// SIMATIC S7-200 project (STEP 7-Micro/WIN), CPU 224 REL 02.00

ORGANIZATION_BLOCK 主程序:OB1
TITLE=---|基于 S7-200 PLC 的步进电机控制系统|---
// 设备启动时，程序利用程序启动标志初始化脉冲输出参数，包括脉冲周期500μs和最大步数429496700。用户可以通过旋转方向开关选择电机的旋转方向，并由电机方向控制输出信号控制（1=逆时针，0=顺时针），但只有在电机停止时，才能改变旋转方向，以确保运行中的稳定性。系统配备了启动按钮和停止按钮来控制电机的运行。按下启动按钮时，若无联锁、电机停止且步数大于1，则通过脉冲输出控制寄存器启动脉冲输出，电机开始运动，同时置位电机运行标志。需要注意的是，脉冲输出的步数必须大于1才能启动电机，以保证有效操作。
// 按下停止按钮后，系统调用停止电机子程序停止脉冲输出并复位标志，同时激活联锁，需松开启动按钮才能解除联锁，确保操作安全。用户还可以通过设置参考点按钮初始化电机位置。按下该按钮时，若电机正在运行，系统会先停止电机，然后通过操作模式选择子程序设置参考点并切换模式。在电机运行时，操作模式保持不变，以维持当前任务的顺利进行。
// 参考点设置完成后，定位控制激活指示点亮，系统进入定位控制模式。此时，用户输入定位角度，定位控制子程序根据角度计算步数（角度/9 * 25 + 余数调整），并由步数调整子程序微调步数，确保定位精度。只有在参考点已设置后，才能执行定位控制，以保证定位的准确性。当脉冲输出完成时，脉冲中止中断自动触发，复位电机运行标志，确保电机及时停止并避免超程。
BEGIN
Network 1 // 网络标题
// 用脉冲输出进行定位控制
LD     SM0.1
R      M0.0, 128             //M0.0 至MD12复位
ATCH   INT_0:INT0, 19
//把中断0分配给中断事件19 (脉冲串终止)
ENI
//脉冲输出功能初始化
MOVW   500, SMW68            //脉冲周期T=500US
MOVW   0, SMW70              // 脉冲宽度为0(脉冲调制)
MOVD   429496700, SMD72      //为参考点设定最大脉冲数
//设置逆时针旋转
LDN    M0.1                  //若电机停止
A      I1.5                  //且旋转主向开关=1 
S      Q0.2, 1               //则逆时针旋转
//设置顺时针旋转
LDN    M0.1                  //若电机停止
AN     I1.5                  //且旋转方向开关=0
R      Q0.2, 1               //则逆时针旋转(Q0.2=0)
//联锁
LD     I1.1
//若按"STOP"(停止)按钮
S      M0.2, 1               //则激活联锁
//解除联锁                   //
LDN    I1.1                  //且"STOP"(停止)按钮松开
AN     I1.0                  //若"START"(启动)按钮松开
R      M0.2, 1               //解除联锁
//确定操作模式(参考点定位控制)
LD     I1.4                  //若按"设置参考点"按钮
EU                           //上升沿
CALL   SBR_1:SBR1
//启动电机
LD     I1.0
// 若按"START"(启动)按钮
EU                           //上升沿
AN     M0.1                  //且电机停止
AN     M0.2                  // 且无联锁
AD>=   SMD72, 1              //且;步数大于1
MOVB   16#85, SMB67          //置脉冲输出功能(PTO)的控制位
PLS    0                     //启动脉冲输出(Q0.0)
S      M0.1, 1               //"电机运行"标志位置位
//定位控制
LD     M0.3                  //若已激活"定位控制"操作模式
AN     M0.1                  //且电机已停止
CALL   SBR_2:SBR2
//停止电机
LD     I1.1                  //若按"STOP"(停止)按钮
EU
A      M0.1                  // 且电机运行
CALL   SBR_0:SBR0
END
END_ORGANIZATION_BLOCK

SUBROUTINE_BLOCK SBR_0:SBR0
TITLE=子程序注释
BEGIN
Network 1 // 网络标题
// 子程序停止电机
MOVB   16#CB, SMB67          //激活脉宽调制
PLS    0                     //停止输出脉冲到Q0.0
R      M0.1, 1               //电机运行标志位复位
CRET                         //子程序结束
END_SUBROUTINE_BLOCK

SUBROUTINE_BLOCK SBR_1:SBR1
TITLE=子程序注释
BEGIN
Network 1 // 网络标题
// 子程序1 "确定操作模式"
LD     M0.1                  // 若电机运行                      // 
CALL   SBR_0:SBR0
//调用子程序0 ,停止电机
//申请参考点曲线
LD     M0.3                  //若已激活"定位控制"则
R      M0.3, 1               //参考点标志位复位(M0.3=0)
R      Q1.0, 1               // 取消"定位控制激活"信息(Q1.0=0)
MOVD   429496700, SMD72      //为新的"参考点曲线"设定最大脉冲数
CRET
//条件返回主程序
//申请定位控制
LDN    M0.3                  //若未设置参考点(M0.3=0),则
S      M0.3, 1               //参考点标志位置位
S      Q1.0, 1               //输出"定位控制激活"信息
CRET
END_SUBROUTINE_BLOCK

SUBROUTINE_BLOCK SBR_2:SBR2
TITLE=子程序注释
BEGIN
Network 1 // 网络标题
// 定位控制
MOVB   IB0, MB11             //把定位角度从IB0 拷到MD8的最低有效字节MB11
R      M8.0, 24              //MB8至MB10清零
DIV    9, MD8                //角度/9 =q1+r1
MOVW   MW8, MW14             //把r1存入MD12
MUL    25, MD8               //q1*25存入MD8
MUL    25, MD12
DIV    9, MD12               //r1*25/9=q2+r2
CALL   SBR_3:SBR3
//在子程序3中循环步数
MOVW   0, MW12               //删除r2
+D     MD12, MD8             //把步数传到MD8
MOVD   MD8, SMD72            //把步数传到SMD72
CRET
END_SUBROUTINE_BLOCK

SUBROUTINE_BLOCK SBR_3:SBR3
TITLE=子程序注释
BEGIN
Network 1 // 网络标题
// 循环步数
LDW>=  MW12, 5               //如果r2>5/0
INCW   MW14                  //步数增加1
CRET
END_SUBROUTINE_BLOCK

INTERRUPT_BLOCK INT_0:INT0
TITLE=中断程序注释
BEGIN
Network 1 // 网络标题
// 脉冲输出中止
R      M0.1, 1               //电机运行标志位复
CRET
Network 5 // 动车辆
END_INTERRUPT_BLOCK
